// TIA Portal V16 export
// export: Created 2025-10-06T17:54:32.6159148Z, ExportSetting WithDefaults, DisplayName Totally Integrated Automation Portal, DisplayVersion V16, DisplayName TIA Portal Version Control Interface, DisplayVersion V16, DisplayName TIA Portal Openness, DisplayVersion V16, DisplayName STEP 7 Professional, DisplayVersion V16, DisplayName STEP 7 Safety, DisplayVersion V16, DisplayName WinCC Advanced, DisplayVersion V16
FUNCTION "EMStopDrives_Block" : Void   // FC14, LAD
VERSION : 0.1
// stored: AutoNumber true, IsIECCheckEnabled false, UDAEnableTagReadback false
   VAR_INPUT
      "Safety Callback" : Bool;
      Direct_Stop : Bool;
   END_VAR
   VAR_OUTPUT
      "Drive 1 Brake Out" : Bool;
      "Drive 2 Brake Out" : Bool;
      "Drive 3 Brake Out" : Bool;
      "Drive 4 Brake Out" : Bool;
      "Drive 5 Brake Out" : Bool;
      "Drive 6 Brake Out" : Bool;
      "Drive 7 Brake Out" : Bool;
      "Drive 8 Brake Out" : Bool;
      "Drive 9 Brake Out" : Bool;
      "Drive 10 Brake Out" : Bool;
   END_VAR
BEGIN

REGION Network 1: Drives Emergency Stop
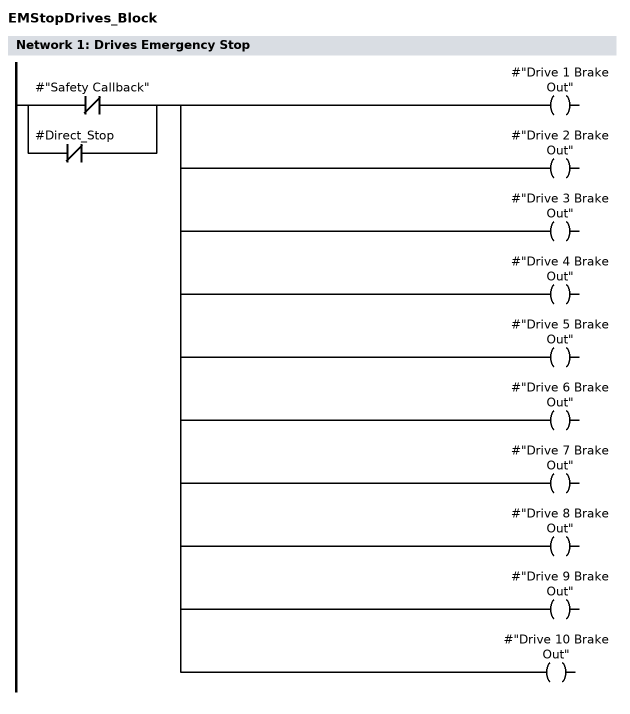
   RUNG wire#powerrail
      I_Contact( #"Safety Callback" )
      wire#w1
      Coil( #"Drive 1 Brake Out" )
   END_RUNG
   RUNG wire#powerrail
      I_Contact( #Direct_Stop )
   END_RUNG wire#w1
   RUNG wire#w1
      Coil( #"Drive 2 Brake Out" )
   END_RUNG
   RUNG wire#w1
      Coil( #"Drive 3 Brake Out" )
   END_RUNG
   RUNG wire#w1
      Coil( #"Drive 4 Brake Out" )
   END_RUNG
   RUNG wire#w1
      Coil( #"Drive 5 Brake Out" )
   END_RUNG
   RUNG wire#w1
      Coil( #"Drive 6 Brake Out" )
   END_RUNG
   RUNG wire#w1
      Coil( #"Drive 7 Brake Out" )
   END_RUNG
   RUNG wire#w1
      Coil( #"Drive 8 Brake Out" )
   END_RUNG
   RUNG wire#w1
      Coil( #"Drive 9 Brake Out" )
   END_RUNG
   RUNG wire#w1
      Coil( #"Drive 10 Brake Out" )
   END_RUNG
   // the same network as SCL:
   #"Drive 1 Brake Out" := NOT #"Safety Callback" OR NOT #Direct_Stop;
   #"Drive 2 Brake Out" := #"Drive 1 Brake Out";
   #"Drive 3 Brake Out" := #"Drive 1 Brake Out";
   #"Drive 4 Brake Out" := #"Drive 1 Brake Out";
   #"Drive 5 Brake Out" := #"Drive 1 Brake Out";
   #"Drive 6 Brake Out" := #"Drive 1 Brake Out";
   #"Drive 7 Brake Out" := #"Drive 1 Brake Out";
   #"Drive 8 Brake Out" := #"Drive 1 Brake Out";
   #"Drive 9 Brake Out" := #"Drive 1 Brake Out";
   #"Drive 10 Brake Out" := #"Drive 1 Brake Out";
END_REGION
END_FUNCTION
